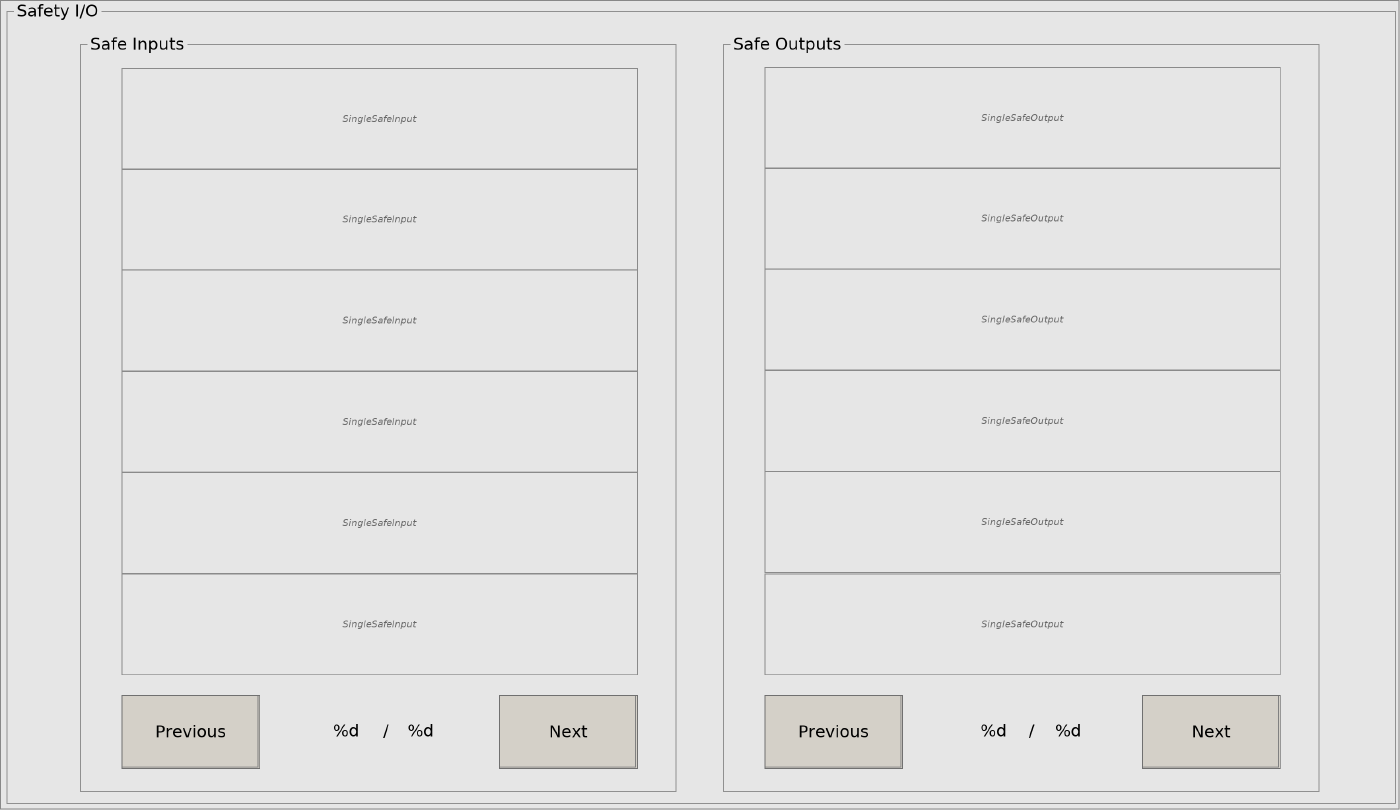
VISUALIZATION PageManualSafety  // 1520x880
VAR_IN_OUT
	btnNextInput			: BOOL;				(*  *)
	btnPreviousInput		: BOOL;				(*  *)
	btnNextOutput			: BOOL;				(*  *)
	btnPreviousOutput		: BOOL;				(*  *)
	
	bNextInvisibleInput		: BOOL;				(*  *)
	bPreviousInvisibleInput	: BOOL;				(*  *)
	bNextInvisibleOutput	: BOOL;				(*  *)
	bPreviousInvisibleOutput: BOOL;				(*  *)	
	
	iSafeInputSelectedPageIndex		: USINT;
	iSafeInputTotalPageIndex 		: USINT;
	iSafeOutputSelectedPageIndex	: USINT;
	iSafeOutputTotalPageIndex 		: USINT;
	
	stSafeOutputEmpty		: ARRAY[1..6] OF BOOL;
	stSafeOutputData		: ARRAY[1..6] OF ST_VisuCtrlOutputFrame;
	stSafeInputEmpty		: ARRAY[1..6] OF BOOL;
	stSafeInputData			: ARRAY[1..6] OF ST_VisuCtrlInputFrame;
END_VAR
    GroupBox (7,4 1508x869), "Safety I/O"
        GroupBox (80,36 647x820), "Safe Inputs"
            Frame (45,583 560x110), invisible if: stSafeInputEmpty[6]
                shows SingleSafeInput(stDigitalInput := stSafeInputData[6])
            Rectangle (345,729 50x50), "%d", text variable: iSafeInputTotalPageIndex+1
            Rectangle (264,729 50x50), "%d", text variable: iSafeInputSelectedPageIndex+1
            Rectangle (1461,1588 130x50), "/"
            Button (45,715 150x80), "Previous", pressed state: btnPreviousInput, invisible if: bPreviousInvisibleInput
                tap btnPreviousInput
            Button (455,715 150x80), "Next", pressed state: btnNextInput, invisible if: bNextInvisibleInput
                tap btnNextInput
            Frame (45,473 560x110), invisible if: stSafeInputEmpty[5]
                shows SingleSafeInput(stDigitalInput := stSafeInputData[5])
            Frame (45,363 560x110), invisible if: stSafeInputEmpty[4]
                shows SingleSafeInput(stDigitalInput := stSafeInputData[4])
            Frame (45,253 560x110), invisible if: stSafeInputEmpty[3]
                shows SingleSafeInput(stDigitalInput := stSafeInputData[3])
            Frame (45,143 560x110), invisible if: stSafeInputEmpty[2]
                shows SingleSafeInput(stDigitalInput := stSafeInputData[2])
            Frame (45,34 560x110), invisible if: stSafeInputEmpty[1]
                shows SingleSafeInput(stDigitalInput := stSafeInputData[1])
            Rectangle (267,729 130x50), "/"
        GroupBox (778,36 647x820), "Safe Outputs"
            Frame (45,583 560x110), invisible if: stSafeOutputEmpty[6]
                shows SingleSafeOutput(stDigitalOutput := stSafeOutputData[6])
            Rectangle (350,729 50x50), "%d", text variable: iSafeOutputTotalPageIndex+1
            Rectangle (269,729 50x50), "%d", text variable: iSafeOutputSelectedPageIndex+1
            Button (45,715 150x80), "Previous", pressed state: btnPreviousOutput, invisible if: bPreviousInvisibleOutput
                tap btnPreviousOutput
            Button (455,715 150x80), "Next", pressed state: btnNextOutput, invisible if: bNextInvisibleOutput
                tap btnNextOutput
            Frame (45,472 560x110), invisible if: stSafeOutputEmpty[5]
                shows SingleSafeOutput(stDigitalOutput := stSafeOutputData[5])
            Frame (45,362 560x110), invisible if: stSafeOutputEmpty[4]
                shows SingleSafeOutput(stDigitalOutput := stSafeOutputData[4])
            Frame (45,252 560x110), invisible if: stSafeOutputEmpty[3]
                shows SingleSafeOutput(stDigitalOutput := stSafeOutputData[3])
            Frame (45,142 560x110), invisible if: stSafeOutputEmpty[2]
                shows SingleSafeOutput(stDigitalOutput := stSafeOutputData[2])
            Frame (45,33 560x110), invisible if: stSafeOutputEmpty[1]
                shows SingleSafeOutput(stDigitalOutput := stSafeOutputData[1])
            Rectangle (270,729 130x50), "/"
END_VISUALIZATION

(* stored: Version 1.1.0.1, ProductVersion 3.1.4024.12
   Visu PageManualSafety: Id {e556d058-89ff-47c9-8fe9-d4a374fd548c} *)
